// Mitsubishi GX Works2 project: 테스트동작   PLC: Q02/Q02H

PROGRAM MAIN
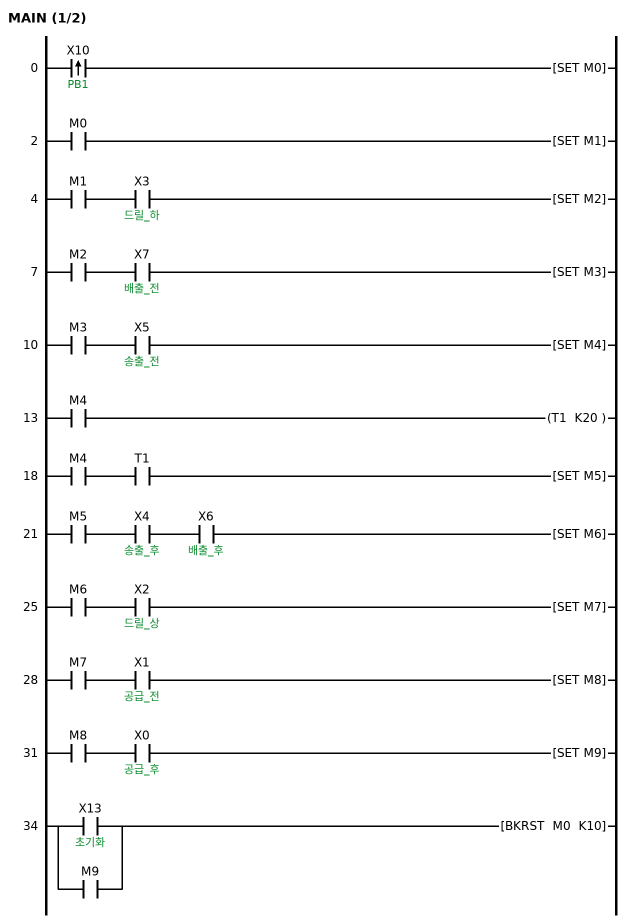
0     LDP     X10  ; PB1
      SET     M0
2     LD      M0
      SET     M1
4     LD      M1
      AND     X3  ; 드릴_하
      SET     M2
7     LD      M2
      AND     X7  ; 배출_전
      SET     M3
10    LD      M3
      AND     X5  ; 송출_전
      SET     M4
13    LD      M4
      OUT     T1 K20
18    LD      M4
      AND     T1
      SET     M5
21    LD      M5
      AND     X4  ; 송출_후
      AND     X6  ; 배출_후
      SET     M6
25    LD      M6
      AND     X2  ; 드릴_상
      SET     M7
28    LD      M7
      AND     X1  ; 공급_전
      SET     M8
31    LD      M8
      AND     X0  ; 공급_후
      SET     M9
34    LD      X13  ; 초기화
      OR      M9
      BKRST   M0 K10
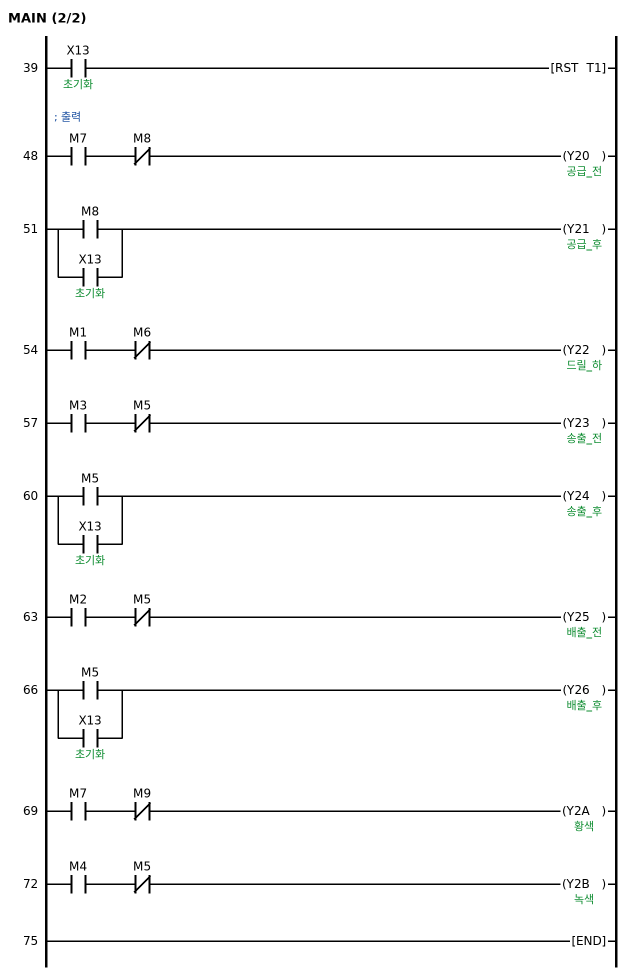
39    LD      X13  ; 초기화
      RST     T1
; 출력
48    LD      M7
      ANI     M8
      OUT     Y20  ; 공급_전
51    LD      M8
      OR      X13  ; 초기화
      OUT     Y21  ; 공급_후
54    LD      M1
      ANI     M6
      OUT     Y22  ; 드릴_하
57    LD      M3
      ANI     M5
      OUT     Y23  ; 송출_전
60    LD      M5
      OR      X13  ; 초기화
      OUT     Y24  ; 송출_후
63    LD      M2
      ANI     M5
      OUT     Y25  ; 배출_전
66    LD      M5
      OR      X13  ; 초기화
      OUT     Y26  ; 배출_후
69    LD      M7
      ANI     M9
      OUT     Y2A  ; 황색
72    LD      M4
      ANI     M5
      OUT     Y2B  ; 녹색
75    END
END_PROGRAM

PROGRAM MAIN1
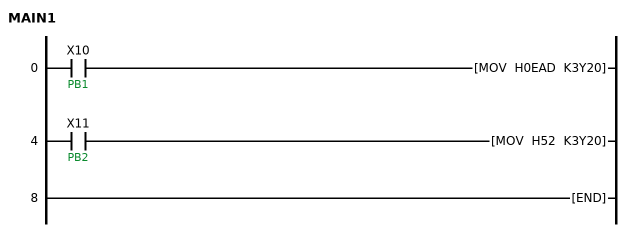
0     LD      X10  ; PB1
      MOV     H0EAD K3Y20  ; 공급_전
4     LD      X11  ; PB2
      MOV     H52 K3Y20
8     END
END_PROGRAM

PROGRAM MAIN2
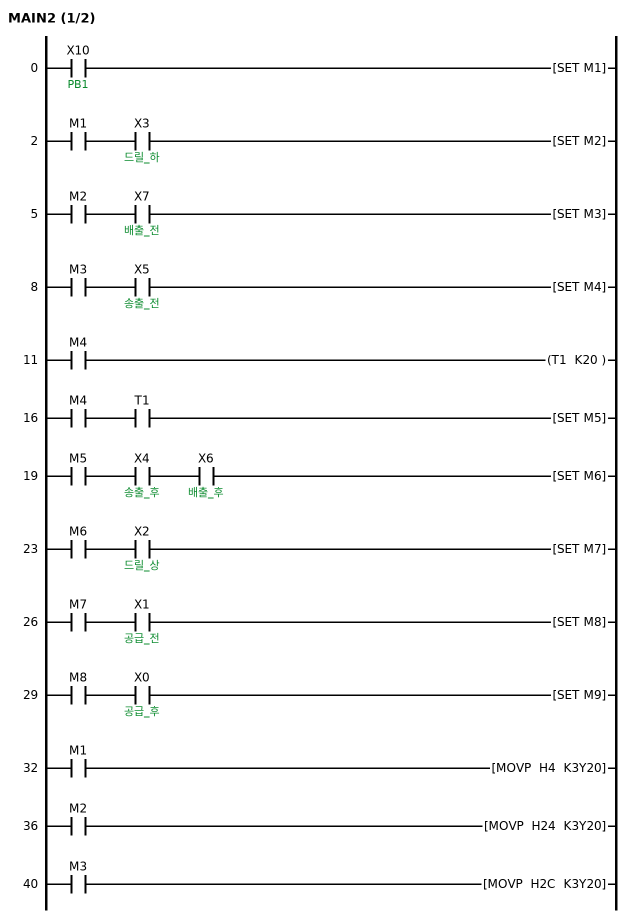
0     LD      X10  ; PB1
      SET     M1
2     LD      M1
      AND     X3  ; 드릴_하
      SET     M2
5     LD      M2
      AND     X7  ; 배출_전
      SET     M3
8     LD      M3
      AND     X5  ; 송출_전
      SET     M4
11    LD      M4
      OUT     T1 K20
16    LD      M4
      AND     T1
      SET     M5
19    LD      M5
      AND     X4  ; 송출_후
      AND     X6  ; 배출_후
      SET     M6
23    LD      M6
      AND     X2  ; 드릴_상
      SET     M7
26    LD      M7
      AND     X1  ; 공급_전
      SET     M8
29    LD      M8
      AND     X0  ; 공급_후
      SET     M9
32    LD      M1
      MOVP    H4 K3Y20  ; 공급_전
36    LD      M2
      MOVP    H24 K3Y20
40    LD      M3
      MOVP    H2C K3Y20
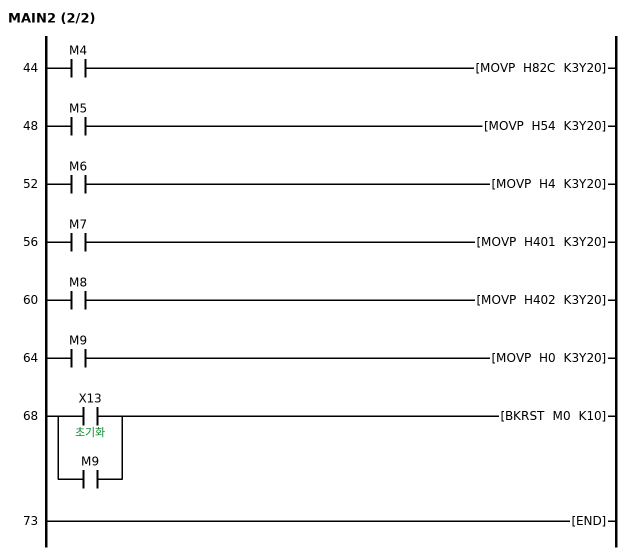
44    LD      M4
      MOVP    H82C K3Y20
48    LD      M5
      MOVP    H54 K3Y20
52    LD      M6
      MOVP    H4 K3Y20
56    LD      M7
      MOVP    H401 K3Y20
60    LD      M8
      MOVP    H402 K3Y20
64    LD      M9
      MOVP    H0 K3Y20
68    LD      X13  ; 초기화
      OR      M9
      BKRST   M0 K10
73    END
END_PROGRAM

// device comments not shown above
X8  ; 메거진
X9  ; 비금속
X0A  ; 금속
X12  ; PB3
Y27  ; 컨베어
Y28  ; 가공드
Y29  ; 적색
